{attribute 'qualified_only'}
{attribute 'strict'}
{attribute 'to_String'}
TYPE eWago750495_MeasureGroupID_1 :
(
	ac := 10,
	harmonicsL1 := 20,
	harmonicsL2 := 21,
	harmonicsL3	:= 22
) USINT;
END_TYPE

(* stored: Version 1.1.0.1, ProductVersion 3.1.4024.12
   DUT eWago750495_MeasureGroupID_1: Id {eabf7032-9b8f-4aea-961c-c835c7719dcd} *)
